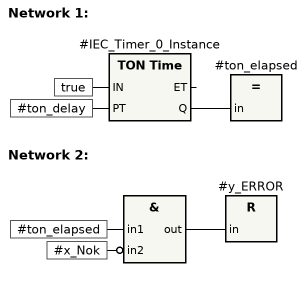
   #IEC_Timer_0_Instance(IN := true, PT := #ton_delay);   // TON
   #ton_elapsed := #IEC_Timer_0_Instance.Q;
END_REGION

REGION Network 2
   IF #ton_elapsed AND NOT #x_Nok THEN #y_ERROR := FALSE; END_IF;
END_REGION
END_FUNCTION_BLOCK

FUNCTION "_buttonsAndLEDs_main" : Void   // FC6, FBD
{ S7_Optimized_Access := 'TRUE' }
VERSION : 0.1
// stored: AutoNumber true, IsIECCheckEnabled false, SetENOAutomatically false, UDAEnableTagReadback false
BEGIN

REGION Network 1
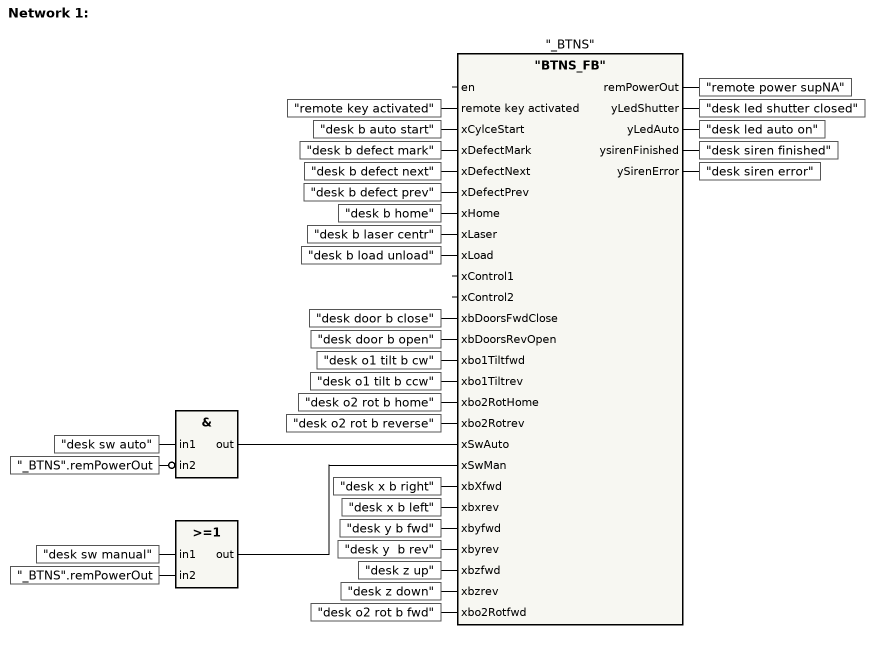
   "_BTNS"("remote key activated" := "remote key activated",   // "BTNS_FB"
           xCylceStart := "desk b auto start",
           xDefectMark := "desk b defect mark",
           xDefectNext := "desk b defect next",
           xDefectPrev := "desk b defect prev",
           xHome := "desk b home",
           xLaser := "desk b laser centr",
           xLoad := "desk b load unload",
           xbDoorsFwdClose := "desk door b close",
           xbDoorsRevOpen := "desk door b open",
           xbo1Tiltfwd := "desk o1 tilt b cw",
           xbo1Tiltrev := "desk o1 tilt b ccw",
           xbo2RotHome := "desk o2 rot b home",
           xbo2Rotrev := "desk o2 rot b reverse",
           xSwAuto := "desk sw auto" AND NOT "_BTNS".remPowerOut,
           xSwMan := "desk sw manual" OR "_BTNS".remPowerOut,
           xbXfwd := "desk x b right",
           xbxrev := "desk x b left",
           xbyfwd := "desk y b fwd",
           xbyrev := "desk y  b rev",
           xbzfwd := "desk z up",
           xbzrev := "desk z down",
           xbo2Rotfwd := "desk o2 rot b fwd",
           remPowerOut => "remote power supNA",
           yLedShutter => "desk led shutter closed",
           yLedAuto => "desk led auto on",
           ysirenFinished => "desk siren finished",
           ySirenError => "desk siren error");
END_REGION
END_FUNCTION

FUNCTION_BLOCK "BTNS_FB"   // FB1, FBD
{ S7_Optimized_Access := 'TRUE' }
VERSION : 0.1
// stored: AutoNumber true, IsIECCheckEnabled false, IsRetainMemResEnabled false, MemoryReserve 100, SetENOAutomatically false, UDAEnableTagReadback false
   VAR_INPUT
      "remote key activated" : Bool;
      xCylceStart : Bool;
      xDefectMark : Bool;
      xDefectNext : Bool;
      xDefectPrev : Bool;
      xHome : Bool;
      xLaser : Bool;
      xLoad : Bool;
      xControl1 : Bool;
      xControl2 : Bool;
      xbDoorsFwdClose : Bool;
      xbDoorsRevOpen : Bool;
      xbo1Tiltfwd : Bool;
      xbo1Tiltrev : Bool;
      xbo2RotHome : Bool;
      xbo2Rotrev : Bool;
      xSwAuto : Bool;
      xSwMan : Bool;
      xbXfwd : Bool;
      xbxrev : Bool;
      xbyfwd : Bool;
      xbyrev : Bool;
      xbzfwd : Bool;
      xbzrev : Bool;
      xbo2Rotfwd : Bool;
   END_VAR
   VAR_OUTPUT
      remPowerOut : Bool;
      yLedShutter : Bool;
      yLedAuto : Bool;
      ysirenFinished : Bool;
      ySirenError : Bool;
   END_VAR
   VAR
      desk_yledShutter { S7_SetPoint := 'True'} : "LED_FBD";
   END_VAR
   VAR_TEMP   // added for the SCL form of the ladder/FBD networks
      _w1 : Bool;
   END_VAR
BEGIN

REGION Network 2
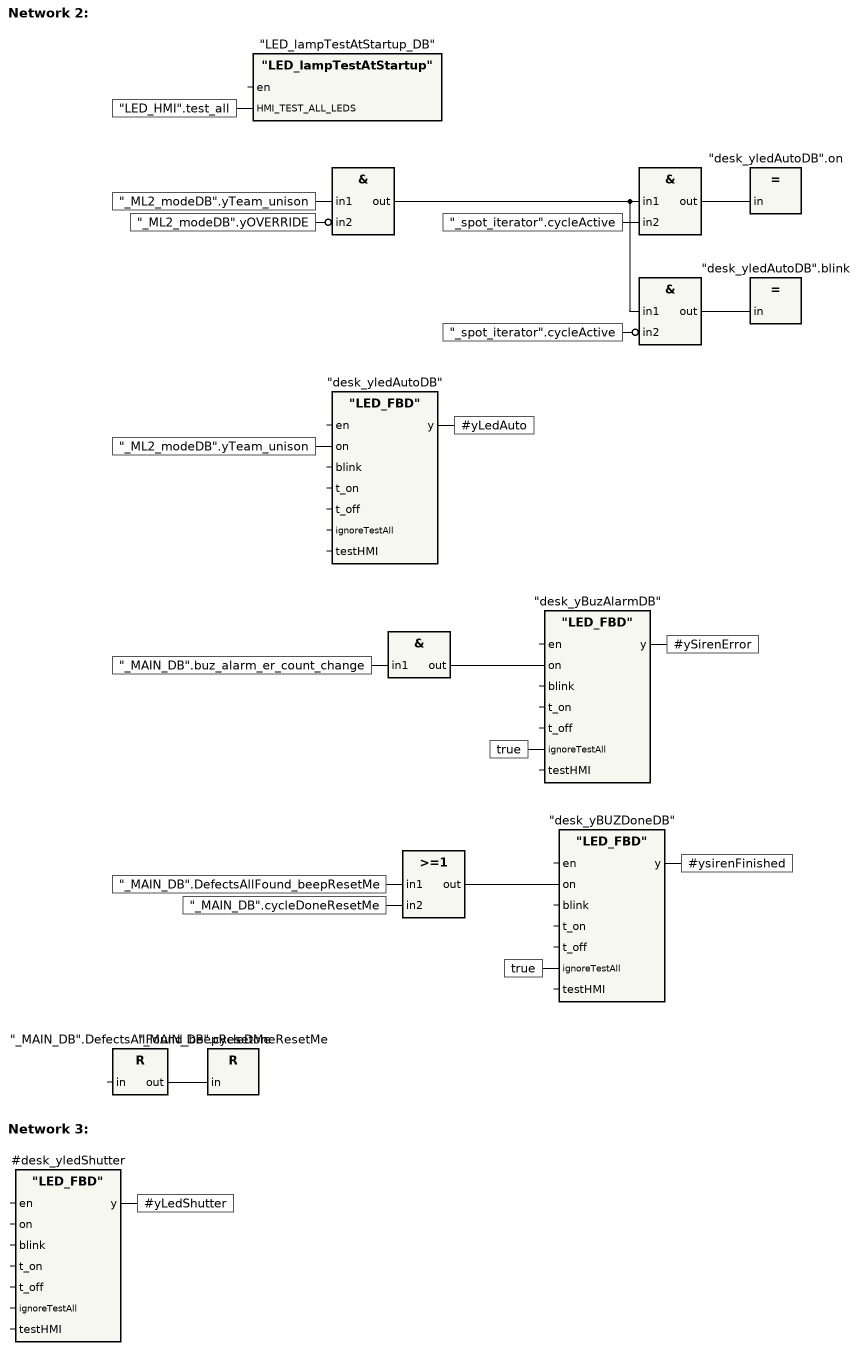
   "LED_lampTestAtStartup_DB"(HMI_TEST_ALL_LEDS := "LED_HMI".test_all);   // "LED_lampTestAtStartup"
   #_w1 := "_ML2_modeDB".yTeam_unison AND NOT "_ML2_modeDB".yOVERRIDE;
   "desk_yledAutoDB".on := #_w1 AND "_spot_iterator".cycleActive;
   "desk_yledAutoDB".blink := #_w1 AND NOT "_spot_iterator".cycleActive;
   "desk_yledAutoDB"(on := "_ML2_modeDB".yTeam_unison, y => #yLedAuto);   // "LED_FBD"
   "desk_yBuzAlarmDB"(on := "_MAIN_DB".buz_alarm_er_count_change, ignoreTestAll := true, y => #ySirenError);   // "LED_FBD"
   "desk_yBUZDoneDB"(on := "_MAIN_DB".DefectsAllFound_beepResetMe OR "_MAIN_DB".cycleDoneResetMe,   // "LED_FBD"
                     ignoreTestAll := true,
                     y => #ysirenFinished);
   "_MAIN_DB".DefectsAllFound_beepResetMe := FALSE;
   "_MAIN_DB".cycleDoneResetMe := FALSE;
END_REGION

REGION Network 3
   #desk_yledShutter(y => #yLedShutter);   // "LED_FBD"
END_REGION

REGION Network 6
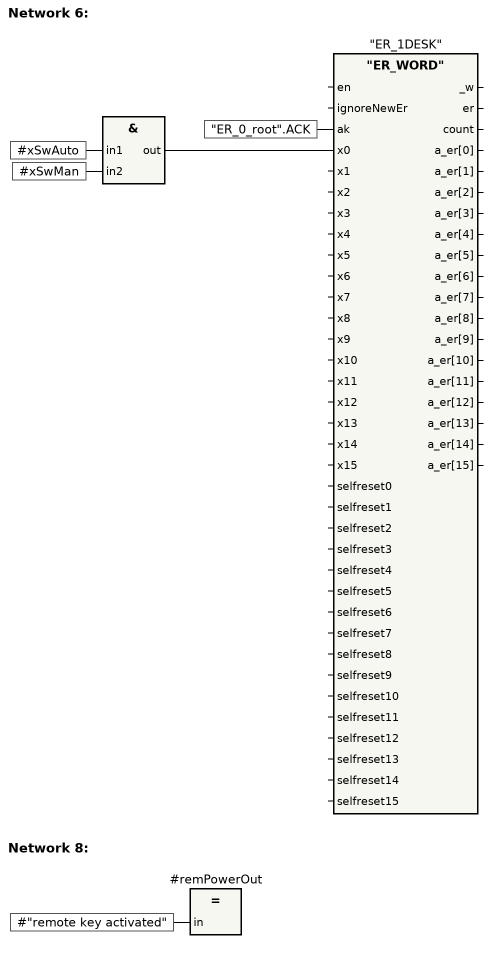
   "ER_1DESK"(ak := "ER_0_root".ACK, x0 := #xSwAuto AND #xSwMan);   // "ER_WORD"
END_REGION

REGION Network 8
   #remPowerOut := #"remote key activated";
END_REGION
END_FUNCTION_BLOCK

FUNCTION_BLOCK "LED_lampTestAtStartup"   // FB43, FBD
{ S7_Optimized_Access := 'TRUE' }
VERSION : 0.1
// stored: AutoNumber true, IsIECCheckEnabled false, IsRetainMemResEnabled false, MemoryReserve 100, SetENOAutomatically false, UDAEnableTagReadback false
   VAR_IN_OUT
      HMI_TEST_ALL_LEDS : Bool;
   END_VAR
   VAR
      IEC_Timer_0_Instance { S7_SetPoint := 'True'} : TON_TIME;
      mem : Bool;
   END_VAR
   VAR_TEMP
      ton_elapsed : Bool;
      trig : Bool;
   END_VAR
   VAR_TEMP   // added for the SCL form of the ladder/FBD networks
      _w1 : Bool;
   END_VAR
BEGIN

REGION Network 1
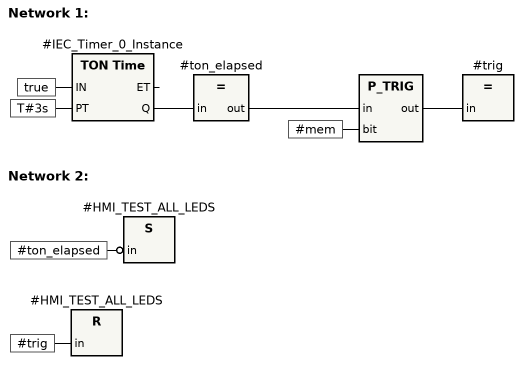
   #IEC_Timer_0_Instance(IN := true, PT := T#3s);   // TON
   #ton_elapsed := #IEC_Timer_0_Instance.Q;
   #_w1 := #IEC_Timer_0_Instance.Q AND NOT #mem;   // rising edge
   #mem := #IEC_Timer_0_Instance.Q;
   #trig := #_w1;
END_REGION

REGION Network 2
   IF NOT #ton_elapsed THEN #HMI_TEST_ALL_LEDS := TRUE; END_IF;
   IF #trig THEN #HMI_TEST_ALL_LEDS := FALSE; END_IF;
END_REGION
END_FUNCTION_BLOCK

FUNCTION_BLOCK "LED_FBD"   // FB54, FBD
{ S7_Optimized_Access := 'TRUE' }
VERSION : 0.1
// stored: AutoNumber true, IsIECCheckEnabled false, IsRetainMemResEnabled false, MemoryReserve 100, SetENOAutomatically false, UDAEnableTagReadback false
   VAR_INPUT
      on : Bool;
      blink : Bool;
      t_on : Time := T#1s;
      t_off : Time := T#1s;
      ignoreTestAll : Bool;
   END_VAR
   VAR_OUTPUT
      y : Bool;
   END_VAR
   VAR_IN_OUT
      testHMI : Bool;
   END_VAR
   VAR
      blink1 { S7_SetPoint := 'True'} : "BLINKER";
      blink_st : Bool;
      tonhmi { S7_SetPoint := 'True'} : TON_TIME;
   END_VAR
BEGIN

REGION Network 1
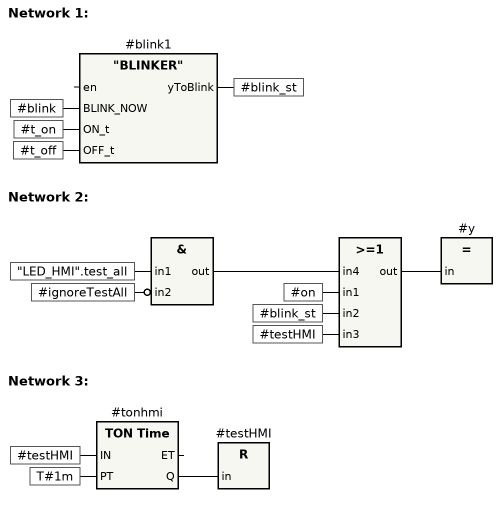
   #blink1(BLINK_NOW := #blink, ON_t := #t_on, OFF_t := #t_off, yToBlink => #blink_st);   // "BLINKER"
END_REGION

REGION Network 2
   #y := ("LED_HMI".test_all AND NOT #ignoreTestAll) OR #on OR #blink_st OR #testHMI;
END_REGION

REGION Network 3
   #tonhmi(IN := #testHMI, PT := T#1m);   // TON
   IF #tonhmi.Q THEN #testHMI := FALSE; END_IF;
END_REGION
END_FUNCTION_BLOCK

FUNCTION "fpd_magnet_lightbarrier_main" : Void   // FC3, FBD
{ S7_Optimized_Access := 'TRUE' }
VERSION : 0.1
// stored: AutoNumber true, IsIECCheckEnabled false, SetENOAutomatically false, UDAEnableTagReadback false
   VAR_TEMP
      er_no_clos : Bool;
      er_no_opn : Bool;
      er_both_sensors : Bool;
   END_VAR
BEGIN

REGION Network 1
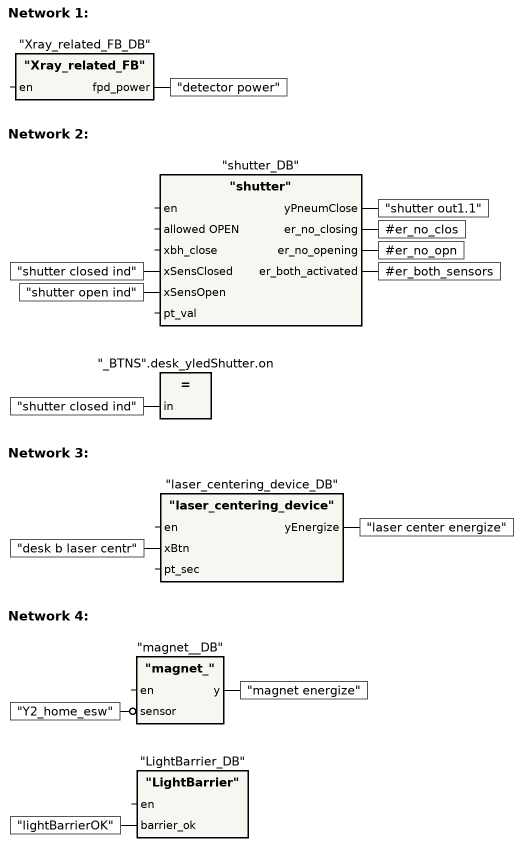
   "Xray_related_FB_DB"(fpd_power => "detector power");   // "Xray_related_FB"
END_REGION

REGION Network 2
   "shutter_DB"(xSensClosed := "shutter closed ind",   // "shutter"
                xSensOpen := "shutter open ind",
                yPneumClose => "shutter out1.1",
                er_no_closing => #er_no_clos,
                er_no_opening => #er_no_opn,
                er_both_activated => #er_both_sensors);
   "_BTNS".desk_yledShutter.on := "shutter closed ind";
END_REGION

REGION Network 3
   "laser_centering_device_DB"(xBtn := "desk b laser centr", yEnergize => "laser center energize");   // "laser_centering_device"
END_REGION

REGION Network 4
   "magnet__DB"(sensor := NOT "Y2_home_esw", y => "magnet energize");   // "magnet_"
   "LightBarrier_DB"(barrier_ok := "lightBarrierOK");   // "LightBarrier"
END_REGION

REGION Network 5
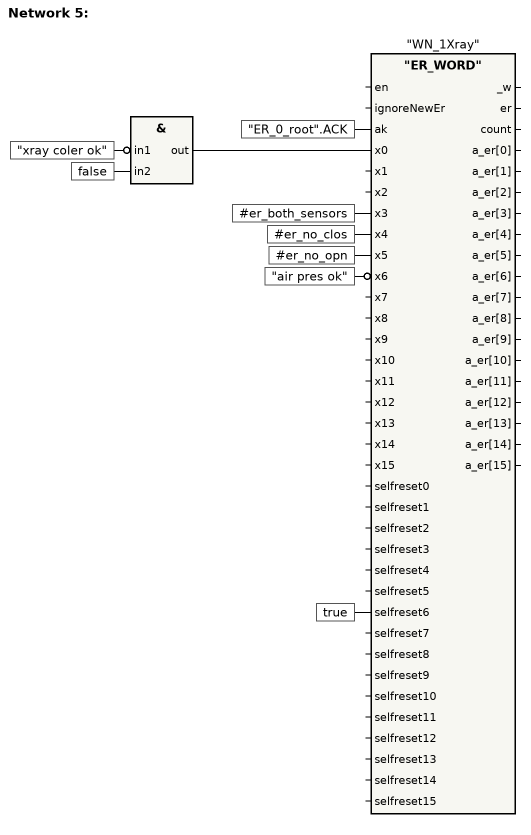
   "WN_1Xray"(ak := "ER_0_root".ACK,   // "ER_WORD"
              x0 := NOT "xray coler ok" AND false,
              x3 := #er_both_sensors,
              x4 := #er_no_clos,
              x5 := #er_no_opn,
              x6 := NOT "air pres ok",
              selfreset6 := true);
END_REGION
END_FUNCTION

FUNCTION_BLOCK "Xray_related_FB"   // FB56, FBD
{ S7_Optimized_Access := 'TRUE' }
VERSION : 0.1
// stored: AutoNumber true, IsIECCheckEnabled false, IsRetainMemResEnabled false, MemoryReserve 100, SetENOAutomatically false, UDAEnableTagReadback false
   VAR_OUTPUT
      fpd_power : Bool;
   END_VAR
BEGIN

REGION Network 1
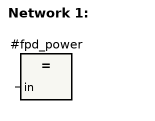
   #fpd_power := TRUE;
END_REGION
END_FUNCTION_BLOCK

FUNCTION_BLOCK "shutter"   // FB42, FBD
{ S7_Optimized_Access := 'TRUE' }
VERSION : 0.1
// stored: AutoNumber true, IsIECCheckEnabled false, IsRetainMemResEnabled false, MemoryReserve 100, SetENOAutomatically false, UDAEnableTagReadback false
   VAR_INPUT
      "allowed OPEN" : Bool := true;
      xbh_close : Bool;
      xSensClosed : Bool;
      xSensOpen : Bool;
      pt_val : Time := T#3s;
   END_VAR
   VAR_OUTPUT
      yPneumClose : Bool;
      er_no_closing : Bool;
      er_no_opening : Bool;
      er_both_activated : Bool;
   END_VAR
   VAR
      tonclos { S7_SetPoint := 'True'} : TON_TIME;
      tonopn { S7_SetPoint := 'True'} : TON_TIME;
   END_VAR
   VAR RETAIN
      commandClose : Bool;
   END_VAR
   VAR
      mem : Bool;
   END_VAR
   VAR_TEMP
      btn_clk : Bool;
   END_VAR
BEGIN

REGION Network 1
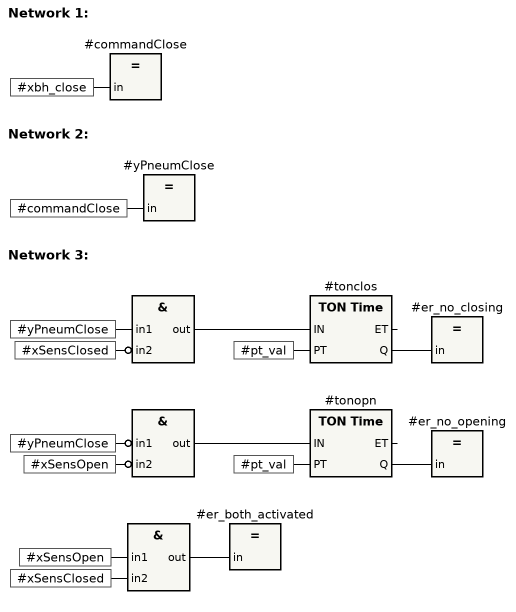
   #commandClose := #xbh_close;
END_REGION

REGION Network 2
   #yPneumClose := #commandClose;
END_REGION

REGION Network 3
   #tonclos(IN := #yPneumClose AND NOT #xSensClosed, PT := #pt_val);   // TON
   #er_no_closing := #tonclos.Q;
   #tonopn(IN := NOT #yPneumClose AND NOT #xSensOpen, PT := #pt_val);   // TON
   #er_no_opening := #tonopn.Q;
   #er_both_activated := #xSensOpen AND #xSensClosed;
END_REGION
END_FUNCTION_BLOCK

FUNCTION_BLOCK "laser_centering_device"   // FB4, FBD
{ S7_Optimized_Access := 'TRUE' }
VERSION : 0.1
// stored: AutoNumber true, IsIECCheckEnabled false, IsRetainMemResEnabled false, MemoryReserve 100, SetENOAutomatically false, UDAEnableTagReadback false
   VAR_INPUT
      xBtn : Bool;
      pt_sec : Real;
   END_VAR
   VAR_OUTPUT
      yEnergize : Bool;
   END_VAR
   VAR RETAIN
      pt : Time := T#10s;
   END_VAR
   VAR
      mem : Bool;
      clkBtn : Bool;
      IEC_Timer_0_Instance { S7_SetPoint := 'True'} : TON_TIME;
      xBtnWAS : Bool;
      should_energize_was : Bool;
   END_VAR
BEGIN

REGION Network 2 (SCL)
   #pt := REAL_TO_DINT(#pt_sec * 1000);


   IF #xBtn AND NOT #xBtnWAS THEN
       IF #yEnergize THEN
           #yEnergize := false;
       ELSE
           #yEnergize := TRUE;
       END_IF;
   END_IF;
   #xBtnWAS := #xBtn;
END_REGION

REGION Network 3
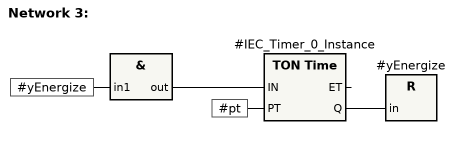
   #IEC_Timer_0_Instance(IN := #yEnergize, PT := #pt);   // TON
   IF #IEC_Timer_0_Instance.Q THEN #yEnergize := FALSE; END_IF;
END_REGION
END_FUNCTION_BLOCK

FUNCTION_BLOCK "magnet_"   // FB71, FBD
{ S7_Optimized_Access := 'TRUE' }
VERSION : 0.1
// stored: AutoNumber true, IsIECCheckEnabled false, IsRetainMemResEnabled false, MemoryReserve 100, SetENOAutomatically false, UDAEnableTagReadback false
   VAR_INPUT
      sensor : Bool;
   END_VAR
   VAR_OUTPUT
      y : Bool;
   END_VAR
   VAR
      energize : Bool;
   END_VAR
   VAR RETAIN
      seconds : Real;
   END_VAR
   VAR
      ton { S7_SetPoint := 'True'} : TON_TIME;
      pt_ms : Time;
   END_VAR
BEGIN

REGION Network 1
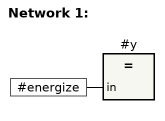
   #y := #energize;
END_REGION

REGION Network 2 (SCL)
   #pt_ms := REAL_TO_DINT(#seconds * 1000.0);
END_REGION
END_FUNCTION_BLOCK

FUNCTION_BLOCK "LightBarrier"   // FB75, FBD
{ S7_Optimized_Access := 'TRUE' }
VERSION : 0.1
// stored: AutoNumber true, IsIECCheckEnabled false, IsRetainMemResEnabled false, MemoryReserve 100, SetENOAutomatically false, UDAEnableTagReadback false
   VAR_INPUT
      barrier_ok : Bool;
   END_VAR
BEGIN
END_FUNCTION_BLOCK

FUNCTION "_coordinate_database_manager_main" : Void   // FC14, FBD
{ S7_Optimized_Access := 'TRUE' }
VERSION : 0.1
// stored: AutoNumber true, IsIECCheckEnabled false, SetENOAutomatically false, UDAEnableTagReadback false
BEGIN

REGION Network 1
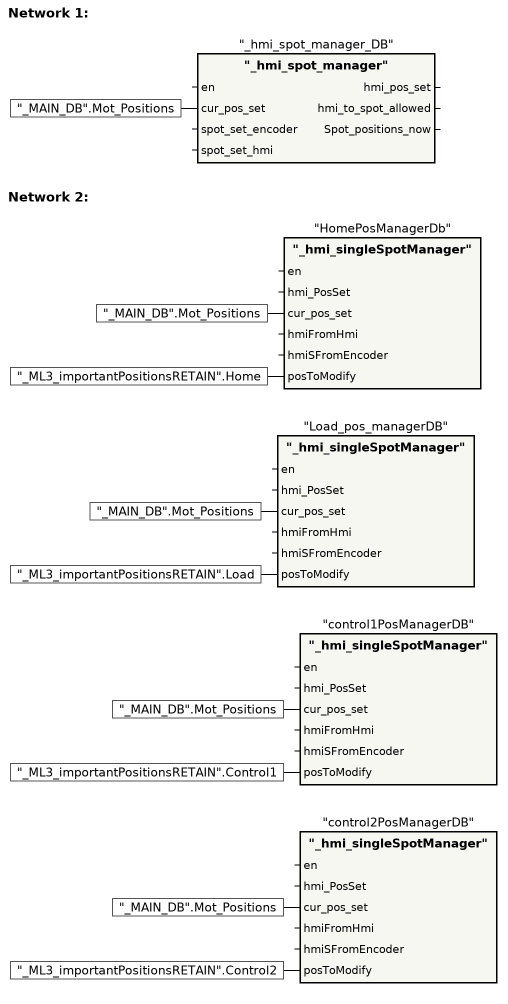
   "_hmi_spot_manager_DB"(cur_pos_set := "_MAIN_DB".Mot_Positions);   // "_hmi_spot_manager"
END_REGION

REGION Network 2
   "HomePosManagerDb"(cur_pos_set := "_MAIN_DB".Mot_Positions,   // "_hmi_singleSpotManager"
                      posToModify := "_ML3_importantPositionsRETAIN".Home);
   "Load_pos_managerDB"(cur_pos_set := "_MAIN_DB".Mot_Positions,   // "_hmi_singleSpotManager"
                        posToModify := "_ML3_importantPositionsRETAIN".Load);
   "control1PosManagerDB"(cur_pos_set := "_MAIN_DB".Mot_Positions,   // "_hmi_singleSpotManager"
                          posToModify := "_ML3_importantPositionsRETAIN".Control1);
   "control2PosManagerDB"(cur_pos_set := "_MAIN_DB".Mot_Positions,   // "_hmi_singleSpotManager"
                          posToModify := "_ML3_importantPositionsRETAIN".Control2);
END_REGION
END_FUNCTION

FUNCTION_BLOCK "_hmi_spot_manager"   // FB47, FBD
{ S7_Optimized_Access := 'TRUE' }
VERSION : 0.1
// stored: AutoNumber true, IsIECCheckEnabled false, IsRetainMemResEnabled false, MemoryReserve 100, SetENOAutomatically false, UDAEnableTagReadback false
   VAR_INPUT
      cur_pos_set : "typePositions";
   END_VAR
   VAR_OUTPUT
      hmi_pos_set : "typePositions";
      hmi_to_spot_allowed : Bool;
      Spot_positions_now : "typePositions";
   END_VAR
   VAR_IN_OUT
      spot_set_encoder : Bool;
      spot_set_hmi : Bool;
   END_VAR
   VAR
      spot_ws : WString;
      part_was : Int;
      spotSaver { S7_SetPoint := 'True'} : "_hmi_singleSpotManager";
   END_VAR
BEGIN

REGION Network 1
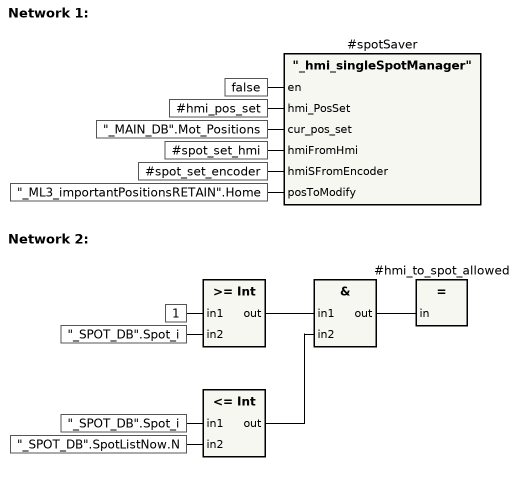
   IF false THEN
       #spotSaver(hmi_PosSet := #hmi_pos_set,   // "_hmi_singleSpotManager"
                  cur_pos_set := "_MAIN_DB".Mot_Positions,
                  hmiFromHmi := #spot_set_hmi,
                  hmiSFromEncoder := #spot_set_encoder,
                  posToModify := "_ML3_importantPositionsRETAIN".Home);
   END_IF;
END_REGION

REGION Network 2
   #hmi_to_spot_allowed := (1 >= "_SPOT_DB".Spot_i) AND ("_SPOT_DB".Spot_i <= "_SPOT_DB".SpotListNow.N);
END_REGION

REGION Network 3 (SCL)
   IF #part_was <> "_SPOT_DB".Part_selected THEN
       IF "_SPOT_DB".Part_selected > 0 AND "_SPOT_DB".Part_selected <= "_SPOT_DB".Spot_N_max THEN
           "_SPOT_DB".SpotListNow := "_SPOT_DB".Parts["_SPOT_DB".Part_selected];
       END_IF;
   ELSE
       IF "_SPOT_DB".Part_selected > 0 AND "_SPOT_DB".Part_selected < "_SPOT_DB".Spot_N_max THEN
           "_SPOT_DB".Parts["_SPOT_DB".Part_selected] := "_SPOT_DB".SpotListNow;
       END_IF;
   END_IF;

   //#Spot_positions_now :=  "_SPOT_DB".SpotListNow.pos_AR["_SPOT_DB".Spot_i];


   #part_was := "_SPOT_DB".Part_selected;
END_REGION
END_FUNCTION_BLOCK

FUNCTION_BLOCK "_hmi_singleSpotManager"   // FB59, FBD
{ S7_Optimized_Access := 'TRUE' }
VERSION : 0.1
// stored: AutoNumber true, IsIECCheckEnabled false, IsRetainMemResEnabled false, MemoryReserve 100, SetENOAutomatically false, UDAEnableTagReadback false
   VAR_INPUT
      hmi_PosSet : "typePositions";
      cur_pos_set : "typePositions";
   END_VAR
   VAR_IN_OUT
      hmiFromHmi : Bool;
      hmiSFromEncoder : Bool;
      posToModify : "typePositions";
   END_VAR
   VAR
      N_max : Int := 99;
   END_VAR
BEGIN

REGION Network 1
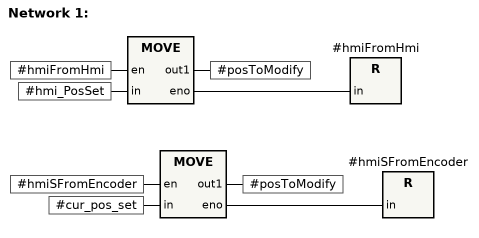
   IF #hmiFromHmi THEN
       #posToModify := #hmi_PosSet;
       #hmiFromHmi := FALSE;
   END_IF;
   IF #hmiSFromEncoder THEN
       #posToModify := #cur_pos_set;
       #hmiSFromEncoder := FALSE;
   END_IF;
END_REGION
END_FUNCTION_BLOCK

FUNCTION "PC_connection_main" : Void   // FC8, FBD
{ S7_Optimized_Access := 'TRUE' }
VERSION : 0.1
// stored: AutoNumber true, IsIECCheckEnabled false, SetENOAutomatically false, UDAEnableTagReadback false
   VAR_TEMP
      er_PC_connection : Bool;
   END_VAR
BEGIN

REGION Network 1
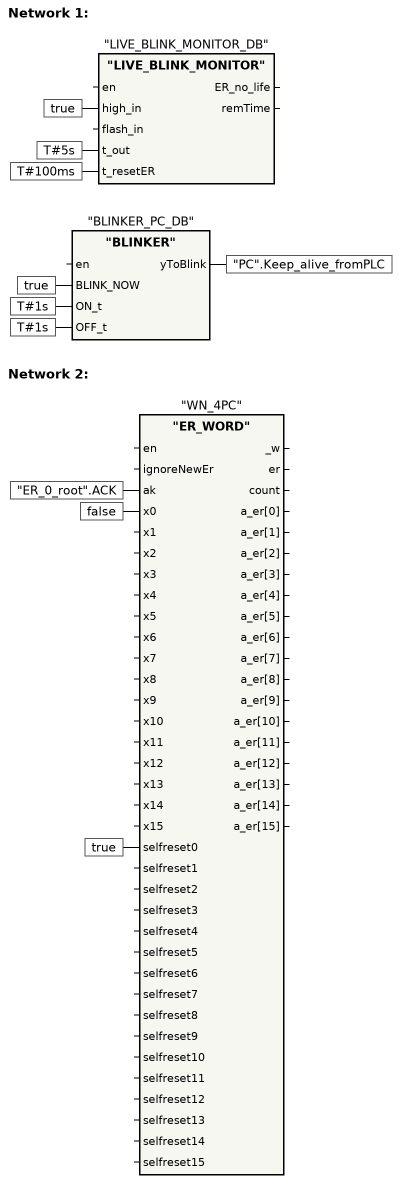
   "LIVE_BLINK_MONITOR_DB"(high_in := true, t_out := T#5s, t_resetER := T#100ms);   // "LIVE_BLINK_MONITOR"
   "BLINKER_PC_DB"(BLINK_NOW := true, ON_t := T#1s, OFF_t := T#1s, yToBlink => "PC".Keep_alive_fromPLC);   // "BLINKER"
END_REGION

REGION Network 2
   "WN_4PC"(ak := "ER_0_root".ACK, x0 := false, selfreset0 := true);   // "ER_WORD"
END_REGION

REGION Network 3
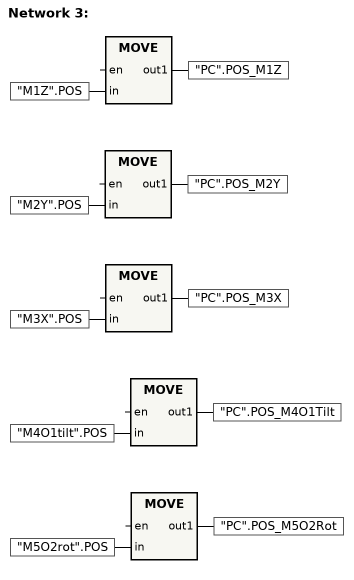
   "PC".POS_M1Z := "M1Z".POS;
   "PC".POS_M2Y := "M2Y".POS;
   "PC".POS_M3X := "M3X".POS;
   "PC".POS_M4O1Tilt := "M4O1tilt".POS;
   "PC".POS_M5O2Rot := "M5O2rot".POS;
END_REGION

REGION Network 4 (SCL)
   %DB69. := %DB69.;
   //%DB69.DBX2.0 := "PC".X_ray_ready_fromPLC;
   //"PC".Image_ready_fromPC := %DB69.DBX4.0;

   IF "PC".PLC_RESET_Image_ready_fromPC THEN
       "PC".Image_ready_fromPC := false;
   END_IF;
END_REGION

REGION Network 6 (SCL)
   (*"PC".POS_M1ZINT := REAL_TO_INT("PC".POS_M1Z);
   "PC".POS_M2YINT := REAL_TO_INT("PC".POS_M2Y);
   "PC".POS_M3XINT := REAL_TO_INT("PC".POS_M3X);
   "PC".POS_M4O1TiltINT := REAL_TO_INT("PC".POS_M4O1TiltINT);
   "PC".POS_M5O2Rot := REAL_TO_INT("PC".POS_M5O2RotINT);*)
END_REGION
END_FUNCTION

FUNCTION_BLOCK "LIVE_BLINK_MONITOR"   // FB65, FBD
{ S7_Optimized_Access := 'TRUE' }
VERSION : 0.1
// stored: AutoNumber true, IsIECCheckEnabled false, IsRetainMemResEnabled false, MemoryReserve 100, SetENOAutomatically false, UDAEnableTagReadback false
   VAR_INPUT
      high_in : Bool;
      flash_in : Bool;
      t_out : Time := T#1s;
      t_resetER : Time := T#5s;
   END_VAR
   VAR_OUTPUT
      ER_no_life : Bool := true;
      remTime : Time;
   END_VAR
   VAR
      tonS { S7_SetPoint := 'True'} : TON_TIME;
      was { S7_SetPoint := 'True'} : Bool;
      tonR { S7_SetPoint := 'True'} : TOF_TIME;
      flashing_ok : Bool;
      flashing_er : Bool;
      high_er : Bool;
   END_VAR
BEGIN

REGION Network 1
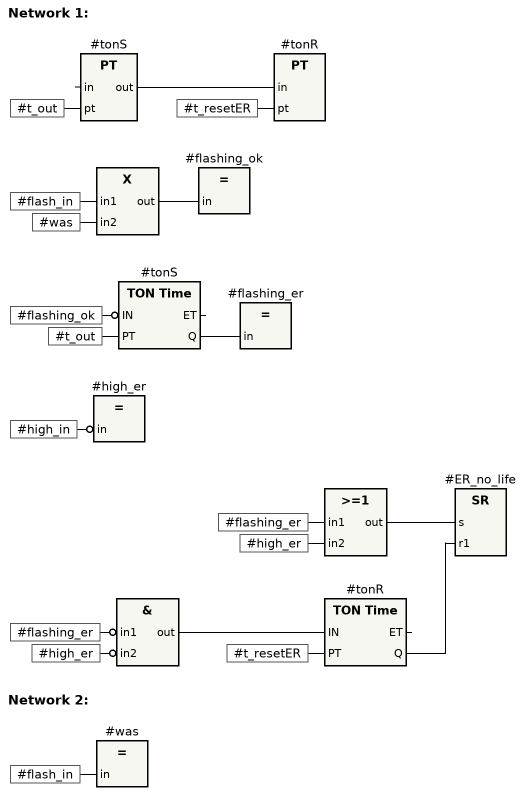
   PRESET_TIMER(PT := #t_out, TIMER := #tonS);
   PRESET_TIMER(PT := #t_resetER, TIMER := #tonR);
   #flashing_ok := #flash_in XOR #was;
   #tonS(IN := NOT #flashing_ok, PT := #t_out);   // TON
   #flashing_er := #tonS.Q;
   #high_er := NOT #high_in;
   #tonR(IN := NOT #flashing_er AND NOT #high_er, PT := #t_resetER);   // TON
   IF #flashing_er OR #high_er THEN
       #ER_no_life := TRUE;   // SR flip-flop
   END_IF;
   IF #tonR.Q THEN #ER_no_life := FALSE; END_IF;
END_REGION

REGION Network 2
   #was := #flash_in;
END_REGION

REGION Network 4 (SCL)
   #remTime := #tonR.PT - #tonR.ET;
END_REGION
END_FUNCTION_BLOCK

FUNCTION "_hmi_main" : Void   // FC26, FBD
{ S7_Optimized_Access := 'TRUE' }
VERSION : 0.1
// stored: AutoNumber true, IsIECCheckEnabled false, SetENOAutomatically false, UDAEnableTagReadback false
BEGIN

REGION Network 1
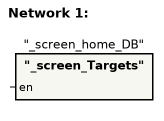
   "_screen_home_DB"();   // "_screen_Targets"
END_REGION
END_FUNCTION

FUNCTION_BLOCK "_screen_Targets"   // FB76, FBD
{ S7_Optimized_Access := 'TRUE' }
VERSION : 0.1
// stored: AutoNumber true, IsIECCheckEnabled false, IsRetainMemResEnabled false, MemoryReserve 100, SetENOAutomatically false, UDAEnableTagReadback false
   VAR
      t_z : "hmi_home_1";
      t_o1 : "hmi_home_1";
      t_o2 : "hmi_home_1";
      t_x : "hmi_home_1";
      t_y : "hmi_home_1";
      z : "hmi_home_1";
      o1 : "hmi_home_1";
      o2 : "hmi_home_1";
      x : "hmi_home_1";
      y : "hmi_home_1";
   END_VAR
BEGIN

REGION Network 1
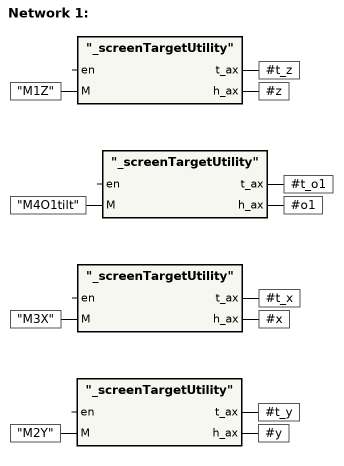
   "_screenTargetUtility"("M" := "M1Z", t_ax => #t_z, h_ax => #z);
   "_screenTargetUtility"("M" := "M4O1tilt", t_ax => #t_o1, h_ax => #o1);
   "_screenTargetUtility"("M" := "M3X", t_ax => #t_x, h_ax => #x);
   "_screenTargetUtility"("M" := "M2Y", t_ax => #t_y, h_ax => #y);
END_REGION

REGION Network 2 (SCL)
   #o2.eF := NOT "M5O2rot".xPredifCal;
   #o2.pos := "M5O2rot".POS;
   #t_o2.pos := "M5O2rot".AMANGRDB.aut_target;
END_REGION
END_FUNCTION_BLOCK

FUNCTION "_screenTargetUtility" : Void   // FC28, FBD
{ S7_Optimized_Access := 'TRUE' }
VERSION : 0.1
// stored: AutoNumber true, IsIECCheckEnabled false, SetENOAutomatically false, UDAEnableTagReadback false
   VAR_INPUT
      "M" : "axis_FBD";
   END_VAR
   VAR_OUTPUT
      t_ax : "hmi_home_1";
      h_ax : "hmi_home_1";
   END_VAR
BEGIN

REGION Network 1 (SCL)
   #h_ax.eF := #M.s_fwd_ind;
   #h_ax.eR := #M.s_rev_ind;
   #h_ax.mF := #M.s_fwd_mechOK;
   #h_ax.mR := #M.s_rev_mecOK;
   #h_ax.pos := #M.POS;

   #t_ax.pos := #M.AMANGRDB.aut_target;
END_REGION
END_FUNCTION

FUNCTION_BLOCK "axis_FBD"   // FB53, FBD
{ S7_Optimized_Access := 'TRUE' }
VERSION : 0.1
// stored: AutoNumber true, IsIECCheckEnabled false, IsRetainMemResEnabled false, MemoryReserve 100, SetENOAutomatically false, UDAEnableTagReadback false
   VAR_INPUT
      "mm_per_ reductur outputshaft_rev (AskURmechEngineer)" : Real := 10.0;
      "reduction_ rotation (AskURmechEngineer)" : Real := 1.0;
      "ABincrements_per_ encoder_rev (CheckEnc Label and HSC hardware settings dont forget input filtration)" : Real := 4096.0;
      "max_revs_ at_10V (CheckMotorLabel)" : Real := 1360.0;
      "enc_placed_ on_motor not reductor output shaft(visually inspect)" : Bool;
      "isMultiturn (visually inspect)" : Bool;
      MultiTurnGoesFwdOnly : Bool;
      soft_speed_change_req : Bool;
      ENC_REVERSED_DIR : Bool;
      ENCODER_DINT : DInt;
      TargetUnison : Real;
      TargetHome : Real;
      Desk_bHome : Bool;
      Desk_bFwd : Bool;
      Desk_bRev : Bool;
      s_fwd_mechOK : Bool;
      s_rev_mecOK : Bool;
      s_fwd_ind : Bool;
      s_rev_ind : Bool;
      xPredifCal : Bool;
      ALIEN_MODE_EN : Bool;
      ALIEN_FWD : Bool;
      ALIEN_REV : Bool;
      ALIEN_SPDABS : Real;
      ExecUni : Bool;
      TheseAreDoors : Bool;
      xOverrideLocal : Bool;
      hbStepPlus : Bool;
      hbStepMinus : Bool;
      TargetStep : Real;
      динамические_границы_используются : Bool;
      динамическая_граница_fwd : Real;
      динамическая_граница_rev : Real;
   END_VAR
   VAR_OUTPUT
      max_speed_10V_p_mm : Real;
      speed_V : Real;
      speed : Real;
      yaINTSPEED : Int;
      yFWD : Bool;
      yREV : Bool;
      yFwd_STOP : Bool;
      yRev_STOP : Bool;
      yIN_POS : Bool;
      ER : Bool;
      WN : Bool;
      ALLOWED : Bool;
      "dist_stop(check t_acc)" : Real;
      MovingHomeWhileFree : Bool;
      ERWSTRING : WString;
   END_VAR
   VAR_IN_OUT
      aut_target : Real;
      para : "typeMotPara";
      POS : Real;
      calibrated : Bool;
      ENC_RET : "typePOSMEMcalib";
   END_VAR
   VAR
      para_ArtLimits { ExternalAccessible := 'False'; ExternalVisible := 'False'; ExternalWritable := 'False'} : "typeMotPara";
      v_absMax : Real;
      au_execute : Bool;
      AMANGRDB { S7_SetPoint := 'True'} : "axis_manager";
      MOTDB { S7_SetPoint := 'True'} : "__mot_universal_";
      WNDB { S7_SetPoint := 'True'} : "ER_WORD";
      ERDB { S7_SetPoint := 'True'} : "ER_WORD";
      erw_calcspd : WString;
      hmiResetCalib : Bool;
      IEC_Timer_0_Instance { S7_SetPoint := 'True'} : TON_TIME;
      artLimiter_Instance { S7_SetPoint := 'True'} : "artLimiter";
   END_VAR
   VAR_TEMP
      counts_per_mm : Real;
      er_params_mech : Bool;
      ENC : DInt;
      selected_man_speed : Real;
      AUTO : Bool;
      MAN : Bool;
      OVERRIDE : Bool;
      counts_real : Real;
      Enc_real_mm : Real;
      er_follow : Bool;
      er_set : Bool;
      er_fwd : Bool;
      er_rev : Bool;
      partners_calibrated : Bool;
      Selected_speed_auto : Real;
      ошибка_динамических_границ : Bool;
   END_VAR
BEGIN

REGION Network 1
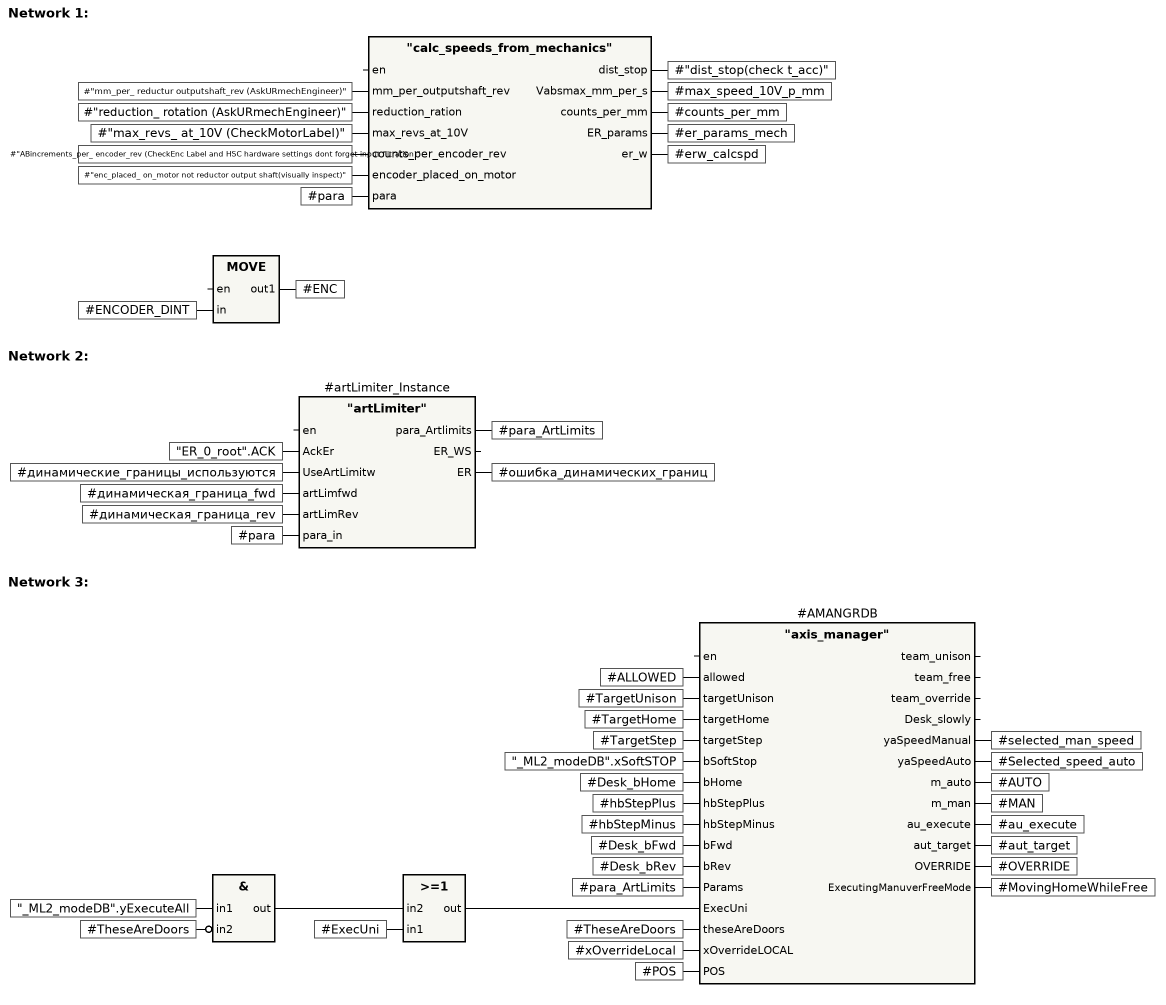
   "calc_speeds_from_mechanics"(mm_per_outputshaft_rev := #"mm_per_ reductur outputshaft_rev (AskURmechEngineer)",
                           reduction_ration := #"reduction_ rotation (AskURmechEngineer)",
                           max_revs_at_10V := #"max_revs_ at_10V (CheckMotorLabel)",
                           counts_per_encoder_rev := #"ABincrements_per_ encoder_rev (CheckEnc Label and HSC hardware settings dont forget input filtration)",
                           encoder_placed_on_motor := #"enc_placed_ on_motor not reductor output shaft(visually inspect)",
                           para := #para,
                           dist_stop => #"dist_stop(check t_acc)",
                           Vabsmax_mm_per_s => #max_speed_10V_p_mm,
                           counts_per_mm => #counts_per_mm,
                           ER_params => #er_params_mech,
                           er_w => #erw_calcspd);
   #ENC := #ENCODER_DINT;
END_REGION

REGION Network 2
   #artLimiter_Instance(AckEr := "ER_0_root".ACK,   // "artLimiter"
                        UseArtLimitw := #динамические_границы_используются,
                        artLimfwd := #динамическая_граница_fwd,
                        artLimRev := #динамическая_граница_rev,
                        para_in := #para,
                        para_Artlimits => #para_ArtLimits,
                        ER => #ошибка_динамических_границ);
END_REGION

REGION Network 3
   #AMANGRDB(allowed := #ALLOWED,   // "axis_manager"
             targetUnison := #TargetUnison,
             targetHome := #TargetHome,
             targetStep := #TargetStep,
             bSoftStop := "_ML2_modeDB".xSoftSTOP,
             bHome := #Desk_bHome,
             hbStepPlus := #hbStepPlus,
             hbStepMinus := #hbStepMinus,
             bFwd := #Desk_bFwd,
             bRev := #Desk_bRev,
             Params := #para_ArtLimits,
             ExecUni := ("_ML2_modeDB".yExecuteAll AND NOT #TheseAreDoors) OR #ExecUni,
             theseAreDoors := #TheseAreDoors,
             xOverrideLOCAL := #xOverrideLocal,
             POS := #POS,
             yaSpeedManual => #selected_man_speed,
             yaSpeedAuto => #Selected_speed_auto,
             m_auto => #AUTO,
             m_man => #MAN,
             au_execute => #au_execute,
             aut_target => #aut_target,
             OVERRIDE => #OVERRIDE,
             ExecutingManuverFreeMode => #MovingHomeWhileFree);
END_REGION

REGION Network 4 (SCL)

   ///1024 ppr, *4* mm per rev /10 reduction = mm
   //
   IF #ENC_REVERSED_DIR THEN
       #counts_real := - DINT_TO_REAL(#ENC);
   ELSE
       #counts_real := + DINT_TO_REAL(#ENC);
   END_IF;


   #Enc_real_mm :=  #counts_real / #counts_per_mm;
END_REGION

REGION Network 5
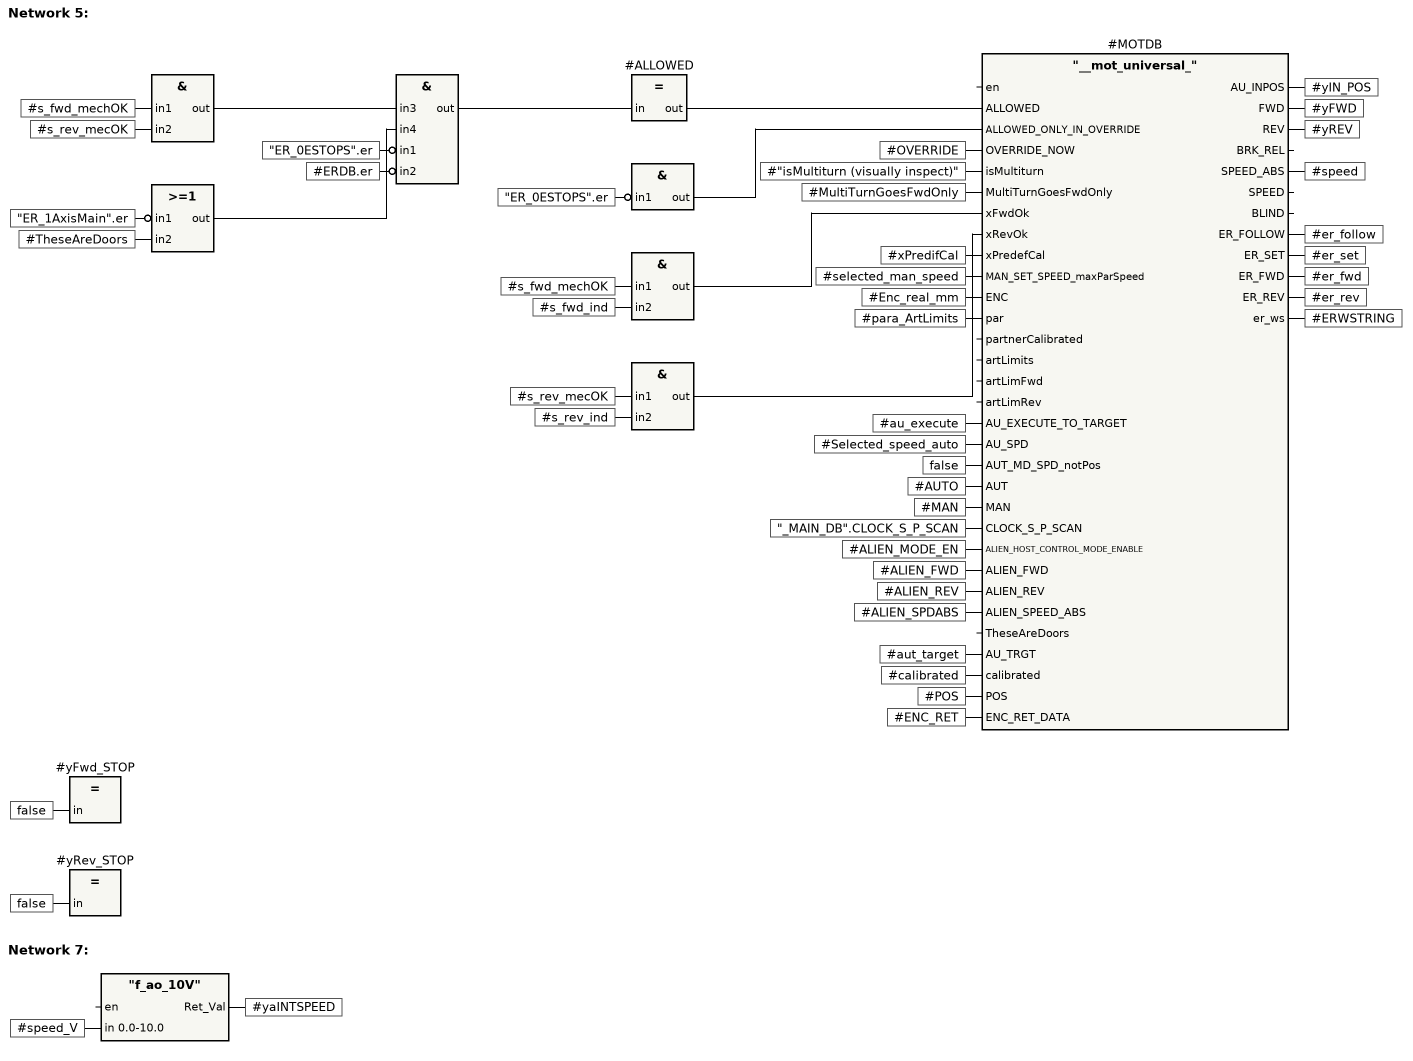
   #ALLOWED := #s_fwd_mechOK AND #s_rev_mecOK AND (NOT "ER_1AxisMain".er OR #TheseAreDoors) AND NOT "ER_0ESTOPS".er AND NOT #ERDB.er;
   #MOTDB(ALLOWED := #ALLOWED,   // "__mot_universal_"
          ALLOWED_ONLY_IN_OVERRIDE := NOT "ER_0ESTOPS".er,
          OVERRIDE_NOW := #OVERRIDE,
          isMultiturn := #"isMultiturn (visually inspect)",
          MultiTurnGoesFwdOnly := #MultiTurnGoesFwdOnly,
          xFwdOk := #s_fwd_mechOK AND #s_fwd_ind,
          xRevOk := #s_rev_mecOK AND #s_rev_ind,
          xPredefCal := #xPredifCal,
          MAN_SET_SPEED_maxParSpeed := #selected_man_speed,
          ENC := #Enc_real_mm,
          par := #para_ArtLimits,
          AU_EXECUTE_TO_TARGET := #au_execute,
          AU_SPD := #Selected_speed_auto,
          AUT_MD_SPD_notPos := false,
          AUT := #AUTO,
          MAN := #MAN,
          CLOCK_S_P_SCAN := "_MAIN_DB".CLOCK_S_P_SCAN,
          ALIEN_HOST_CONTROL_MODE_ENABLE := #ALIEN_MODE_EN,
          ALIEN_FWD := #ALIEN_FWD,
          ALIEN_REV := #ALIEN_REV,
          ALIEN_SPEED_ABS := #ALIEN_SPDABS,
          AU_TRGT := #aut_target,
          calibrated := #calibrated,
          POS := #POS,
          ENC_RET_DATA := #ENC_RET,
          AU_INPOS => #yIN_POS,
          FWD => #yFWD,
          REV => #yREV,
          SPEED_ABS => #speed,
          ER_FOLLOW => #er_follow,
          ER_SET => #er_set,
          ER_FWD => #er_fwd,
          ER_REV => #er_rev,
          er_ws => #ERWSTRING);
   #yFwd_STOP := false;
   #yRev_STOP := false;
END_REGION

REGION Network 6 (SCL)
   #speed_V := #speed / #max_speed_10V_p_mm * 10.0;
END_REGION

REGION Network 7
   #yaINTSPEED := "f_ao_10V"("in 0.0-10.0" := #speed_V);
END_REGION

REGION Network 8
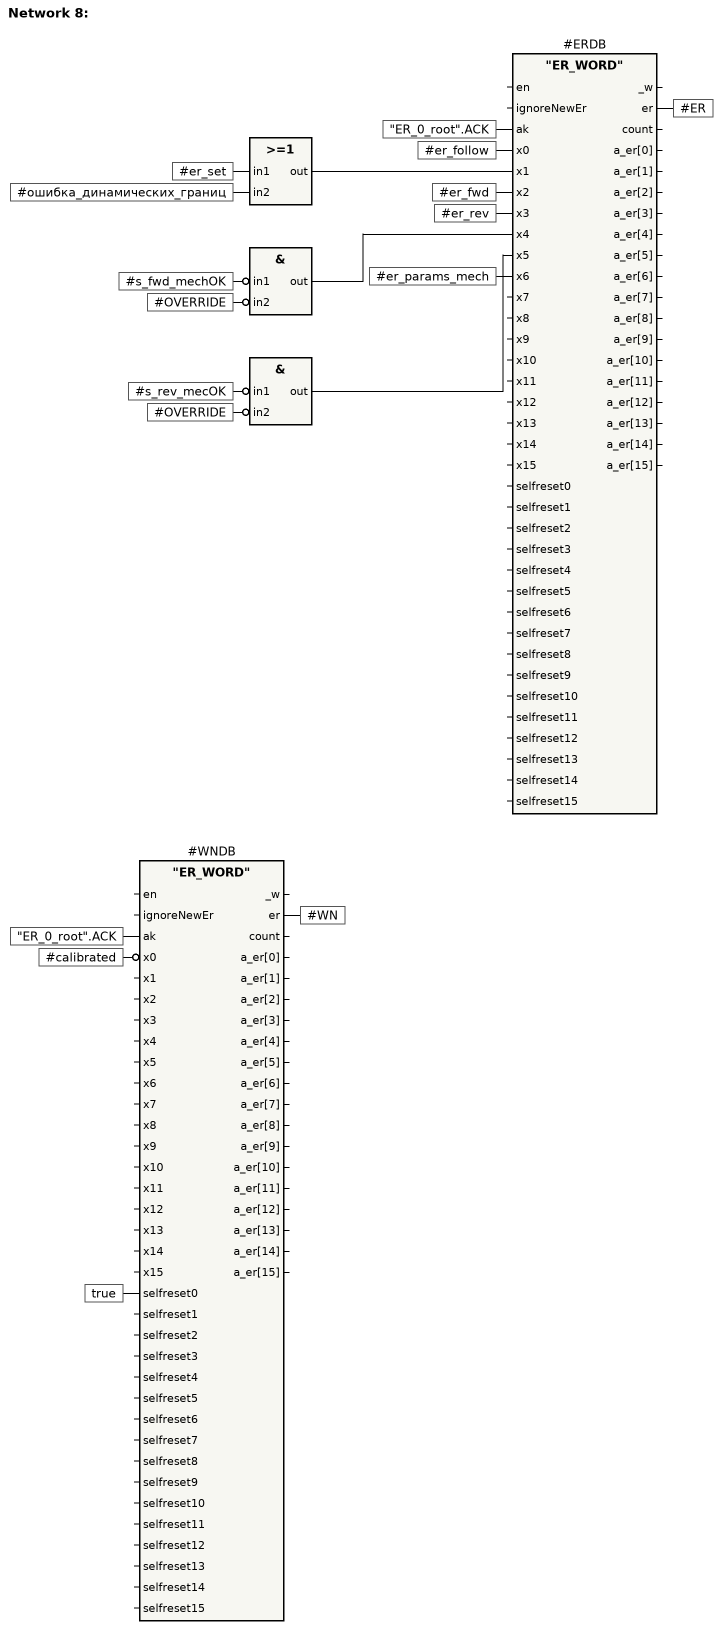
   #ERDB(ak := "ER_0_root".ACK,   // "ER_WORD"
         x0 := #er_follow,
         x1 := #er_set OR #ошибка_динамических_границ,
         x2 := #er_fwd,
         x3 := #er_rev,
         x4 := NOT #s_fwd_mechOK AND NOT #OVERRIDE,
         x5 := NOT #s_rev_mecOK AND NOT #OVERRIDE,
         x6 := #er_params_mech,
         er => #ER);
   #WNDB(ak := "ER_0_root".ACK, x0 := NOT #calibrated, selfreset0 := true, er => #WN);   // "ER_WORD"
END_REGION

REGION Network 9
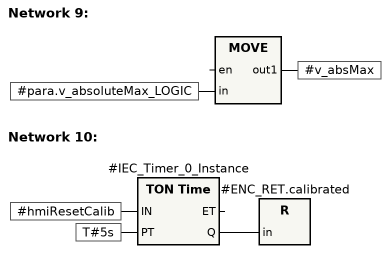
   #v_absMax := #para.v_absoluteMax_LOGIC;
END_REGION

REGION Network 10
   #IEC_Timer_0_Instance(IN := #hmiResetCalib, PT := T#5s);   // TON
   IF #IEC_Timer_0_Instance.Q THEN #ENC_RET.calibrated := FALSE; END_IF;
END_REGION
END_FUNCTION_BLOCK

FUNCTION "calc_speeds_from_mechanics" : Void   // FC15, FBD
{ S7_Optimized_Access := 'TRUE' }
VERSION : 0.1
// stored: AutoNumber true, IsIECCheckEnabled false, SetENOAutomatically false, UDAEnableTagReadback false
   VAR_INPUT
      mm_per_outputshaft_rev : Real;
      reduction_ration : Real;
      max_revs_at_10V : Real;
      counts_per_encoder_rev : Real;
      encoder_placed_on_motor : Bool;
   END_VAR
   VAR_OUTPUT
      dist_stop : Real;
      Vabsmax_mm_per_s : Real;
      counts_per_mm : Real;
      ER_params : Bool;
      er_w : WString;
   END_VAR
   VAR_IN_OUT
      para : "typeMotPara";
   END_VAR
   VAR_TEMP
      t_acceleration_s : Real;
      maxV_mm_per_min : Real;
      "a" : Real;
      v_abs_max : Real;
      dist_auto_done : Real;
      dist_absMax : Real;
      ER_param_1 : Bool;
      ER_param_2 : Bool;
      ER_param_3 : Bool;
      v_crawl : Real;
      t_mx : Real;
   END_VAR
   VAR CONSTANT
      erws1 : WString := WSTRING#'#t_acceleration_s = 0';
      erws2 : WString := WSTRING#'#v_abs_max = 0';
      erws3 : WString := WSTRING#'#t_mx =0';
   END_VAR
BEGIN

REGION Network 1 (SCL)

   #maxV_mm_per_min := #max_revs_at_10V / #reduction_ration * #mm_per_outputshaft_rev;

   #Vabsmax_mm_per_s := #maxV_mm_per_min / 60;
END_REGION

REGION Network 2 (SCL)
   IF #encoder_placed_on_motor THEN
       #counts_per_mm :=  #counts_per_encoder_rev * #reduction_ration / #mm_per_outputshaft_rev  ;
   ELSE
       #counts_per_mm := #counts_per_encoder_rev /  #mm_per_outputshaft_rev;

   END_IF;
END_REGION

REGION Network 4 (SCL)
   #v_crawl := #para.v_crawl_USER;

   #dist_stop:=#para.dist_stop_USER;
   #v_abs_max := #Vabsmax_mm_per_s;
   #para.v_absoluteMax_LOGIC := #v_abs_max;

   #t_mx := #t_acceleration_s := #para.t_acc_50Hz_USER;//:= #t_acc_50Hz_USER;
END_REGION

REGION Network 5 (SCL)
   #er_w := WSTRING#'no er';
   #ER_param_1 := #t_acceleration_s = 0;

   IF #ER_param_1 THEN
       #er_w := #erws1;
   END_IF;


   #ER_param_2 := #v_abs_max = 0;
   IF #ER_param_2 THEN
       #er_w := #erws2;
   END_IF;





   #ER_params := #ER_param_1 OR #ER_param_2 OR #ER_param_3;
END_REGION

REGION Network 6 (SCL)

   IF NOT #ER_params THEN
       #a := (#v_abs_max - #v_crawl) / #t_mx;
       #dist_absMax := #a * #t_mx * #t_mx / 2 + #v_crawl * #t_mx;
   ELSE
       #a := 0;
       #dist_absMax := 999;
   END_IF;
END_REGION

REGION Network 8 (SCL)

   #dist_auto_done := #dist_stop * 3;


   #para.dist_absMax_LOGIC := #dist_absMax;
   #para.dist_auto_done_LOGIC := #dist_auto_done;
   #para.v_auto_USER := LIMIT(MN := 0.0, IN := #para.v_auto_USER, MX := #v_abs_max);
   #para.v_manual_USER := LIMIT(MN := 0.0, IN := #para.v_manual_USER, MX := #v_abs_max);
END_REGION
END_FUNCTION

FUNCTION_BLOCK "artLimiter"   // FB73, FBD
{ S7_Optimized_Access := 'TRUE' }
VERSION : 0.1
// stored: AutoNumber true, IsIECCheckEnabled false, IsRetainMemResEnabled false, MemoryReserve 100, SetENOAutomatically false, UDAEnableTagReadback false
   VAR_INPUT
      AckEr : Bool;
      UseArtLimitw : Bool;
      artLimfwd : Real;
      artLimRev : Real;
      para_in : "typeMotPara";
   END_VAR
   VAR_OUTPUT
      para_Artlimits : "typeMotPara";
      ER_WS : WString;
      ER : Bool;
   END_VAR
   VAR CONSTANT
      ER_WSlimfwdrev : WString := WSTRING#'art lim rev>fwd';
   END_VAR
BEGIN

REGION Network 1
